Yaskawa INFORM job: R2_W72(-45,-90)AWOK.JBI

/JOB
//NAME R2_W72(-45,-90)AWOK
///FOLDERNAME AWOK
//POS
///NPOS 49,49,0,3,0,0
///TOOL 0
///POSTYPE PULSE
///PULSE
C00000=38658,73503,51305,13252,90001,29614
C00001=65523,26705,6655,-13106,85208,4911
C00002=107670,17970,6436,-3368,71268,-84460
C00003=107652,18775,11341,-3415,68666,-84393
C00004=107423,16216,11848,-3383,67035,-84428
C00005=107510,17738,13983,-3423,66508,-84381
C00006=107644,19198,13406,-3437,67615,-84365
C00007=105864,18950,14991,-2899,66440,-84981
C00008=105786,18051,14668,-2879,66175,-85004
C00009=107638,19551,14976,-3454,66830,-84344
C00010=107646,19083,12865,-3431,67888,-84372
C00011=107665,18172,7853,-3381,70500,-84440
C00012=107329,14782,-7472,-3166,78164,78949
C00013=107330,14705,-3413,-3195,75631,79014
C00014=107228,13360,-2084,-3185,74119,79019
C00015=107298,14404,-556,-3212,73719,79054
C00016=107330,14766,-1706,-3209,74613,79041
C00017=107372,15462,-55,-3230,73955,79074
C00018=107289,14311,-411,-3211,73580,79055
C00019=107329,14769,-1561,-3210,74526,79043
C00020=107333,14883,-471,-3220,73914,79061
C00021=107047,14897,3200,-3167,71654,79019
C00022=106435,14835,3634,-2983,71333,78810
C00023=107333,15238,3155,-3253,71868,79115
C00024=107333,14883,-471,-3220,73914,79061
C00025=107330,14766,-1706,-3209,74613,79041
C00026=107330,14705,-3413,-3195,75631,79014
C00027=100153,28277,550,-5705,79007,75993
C00028=100153,27887,7605,-5801,74487,76204
C00029=107294,22988,7404,-8118,72722,78798
C00030=107334,22018,6550,-8130,72754,78811
C00031=107440,25166,9559,-8172,72533,78863
C00032=107023,14605,2817,-11677,68457,74807
C00033=107194,14536,2804,-11739,68452,74869
C00034=107272,14744,5152,-11872,67155,75033
C00035=109703,9347,4240,-12926,65365,76135
C00036=107336,15406,4116,-12788,67547,73901
C00037=107337,14954,-210,-12591,69921,73644
C00038=112500,13425,-9878,-17180,79722,-74576
C00039=112485,14733,7938,-17950,69883,-73131
C00040=111969,16057,13283,-18104,67283,-72919
C00041=111296,15753,14826,-18052,66081,-72985
C00042=111800,14785,12888,-18108,66854,-72915
C00043=111841,17958,15807,-18141,66705,-72876
C00044=106151,16235,9688,-16123,68264,-75269
C00045=107338,15945,7393,-16354,69717,-75029
C00046=107338,15248,2657,-16122,72176,-75369
C00047=107337,15744,-13503,-15550,82007,-76656
C00048=107340,15974,-13399,-15549,82062,-76661
BC00000=89471,358308,1075162
BC00001=68407,333287,1075165
BC00002=10055,263972,1075175
BC00003=10767,263961,1075175
BC00004=11308,262543,1075175
BC00005=11308,262543,1075175
BC00006=11053,263956,1075175
BC00007=11110,264196,1075175
BC00008=11110,264196,1075175
BC00009=11110,264196,1075175
BC00010=10825,264200,1075175
BC00011=10112,264212,1075175
BC00012=140937,263885,1075175
BC00013=141696,263919,1075175
BC00014=142236,262660,1075175
BC00015=142236,262660,1075175
BC00016=141999,263933,1075175
BC00017=143361,264733,1075175
BC00018=143361,264733,1075175
BC00019=143340,263102,1075175
BC00020=126626,262039,1075175
BC00021=126734,267843,1075175
BC00022=126734,267843,1075175
BC00023=126734,267843,1075175
BC00024=126626,262039,1075175
BC00025=141999,263933,1075175
BC00026=141696,263919,1075175
BC00027=128122,271633,1075175
BC00028=128122,271633,1075175
BC00029=155211,273762,1075175
BC00030=129858,271740,1075175
BC00031=129858,271740,1075175
BC00032=122568,266668,1075175
BC00033=122568,266668,1075175
BC00034=113555,268823,1075175
BC00035=113554,268822,1075171
BC00036=110383,269646,1075175
BC00037=107709,269889,1075175
BC00038=15,258637,1075175
BC00039=15,258642,1075175
BC00040=15,258731,1075175
BC00041=15,258766,1075175
BC00042=15,258766,1075175
BC00043=15,258766,1075175
BC00044=99510,267713,1075175
BC00045=101317,267892,1075175
BC00046=99872,267803,1075175
BC00047=99830,267798,1075175
BC00048=99830,440218,1075171
///POSTYPE BASE
///RECTAN
///RCONF 0,0,0,0,0,0,0,0,0,0,0,0,0,0,0,0,0,0,0,0,0,0,0,0
P00006=0.222,-3.123,-1.508,0.0000,0.0000,0.0000
P00021=-0.225,-6.128,-0.405,0.0000,0.0000,0.0000
P00022=0.222,-3.123,-1.508,0.0000,0.0000,0.0000
//INST
///DATE 2023/11/16 10:50
///ATTR SC,RW
///GROUP1 RB1,BS1
NOP
'r2_W72(-45,-90)
'Path S809
SFTOF
MOVJ C00000 BC00000 VJ=20.00
MOVJ C00001 BC00001 VJ=20.00
MOVL C00002 BC00002 V=100.0
MOVL C00003 BC00003 V=100.0
MOVL C00004 BC00004 V=60.0
REFP 3 C00005 BC00005
CALL JOB:SEARCH-R1
SET P022 P006
SFTON P022
MOVL C00006 BC00006 V=60.0
MOVL C00007 BC00007 V=60.0
REFP 3 C00008 BC00008
CALL JOB:SEARCH-R1
SET P022 P006
SFTON P022
MOVL C00009 BC00009 V=60.0
MOVL C00010 BC00010 V=100.0
MOVL C00011 BC00011 V=100.0
'Path S813
SFTOF
MOVJ C00012 BC00012 VJ=20.00
MOVL C00013 BC00013 V=100.0
MOVL C00014 BC00014 V=60.0
REFP 3 C00015 BC00015
CALL JOB:SEARCH-R1
SET P021 P006
SFTON P021
MOVL C00016 BC00016 V=60.0
MOVL C00017 BC00017 V=60.0
REFP 3 C00018 BC00018
CALL JOB:SEARCH-R1
SET P021 P006
SFTON P021
MOVL C00019 BC00019 V=60.0
MOVL C00020 BC00020 V=100.0
MOVL C00021 BC00021 V=60.0
REFP 3 C00022 BC00022
CALL JOB:SEARCH-R1
SET P021 P006
SFTON P021
MOVL C00023 BC00023 V=60.0
MOVL C00024 BC00024 V=100.0
MOVL C00025 BC00025 V=100.0
MOVL C00026 BC00026 V=100.0
'Path W108
SFTOF
SFTON P021
MOVJ C00027 BC00027 VJ=20.00
MOVL C00028 BC00028 V=100.0
MOVL C00029 BC00029 V=100.0 PL=0
REFP 1 C00030 BC00030
REFP 2 C00031 BC00031
MACRO1 MJ#(0) ARGF9
ARCON
MOVL C00032 BC00032 V=11.7
MOVL C00033 BC00033 V=10.8
MOVL C00034 BC00034 V=10.8
MOVL C00035 BC00035 V=10.8
ARCOF
MOVL C00036 BC00036 V=100.0
MOVL C00037 BC00037 V=100.0
SFTOF
'Path W110
SFTOF
SFTON P022
MOVJ C00038 BC00038 VJ=20.00
MOVJ C00039 BC00039 VJ=20.00
MOVL C00040 BC00040 V=100.0
MOVL C00041 BC00041 V=100.0 PL=0
REFP 1 C00042 BC00042
REFP 2 C00043 BC00043
MACRO1 MJ#(0) ARGF9
ARCON
SFTON P021
MOVL C00044 BC00044 V=10.8
ARCOF
MOVL C00045 BC00045 V=100.0
MOVL C00046 BC00046 V=100.0
MOVL C00047 BC00047 V=100.0
SFTOF
MOVJ C00048 BC00048 VJ=20.00
END
